(* IEC 61131-3 sources: TA/Tests/RetainTest/FB (part 2) *)

    AUTO1_OUT_ULINT[0] := AUTO1_OUT_ULINT[0] + 1;
    AUTO1_OUT_ULINT[1] := AUTO1_OUT_ULINT[1] + 1;
    AUTO1_OUT_ULINT[2] := AUTO1_OUT_ULINT[2] + 1;
    AUTO1_OUT_ULINT[3] := AUTO1_OUT_ULINT[3] + 1;
    AUTO1_OUT_ULINT[4] := AUTO1_OUT_ULINT[4] + 1;
    AUTO1_OUT_ULINT[5] := AUTO1_OUT_ULINT[5] + 1;
    AUTO1_OUT_ULINT[6] := AUTO1_OUT_ULINT[6] + 1;
    AUTO1_OUT_ULINT[7] := AUTO1_OUT_ULINT[7] + 1;
    AUTO1_OUT_ULINT[8] := AUTO1_OUT_ULINT[8] + 1;
    AUTO1_OUT_ULINT[9] := AUTO1_OUT_ULINT[9] + 1;

    AUTO1_OUT_USINT[0] := AUTO1_OUT_USINT[0] + 1;
    AUTO1_OUT_USINT[1] := AUTO1_OUT_USINT[1] + 1;
    AUTO1_OUT_USINT[2] := AUTO1_OUT_USINT[2] + 1;
    AUTO1_OUT_USINT[3] := AUTO1_OUT_USINT[3] + 1;
    AUTO1_OUT_USINT[4] := AUTO1_OUT_USINT[4] + 1;
    AUTO1_OUT_USINT[5] := AUTO1_OUT_USINT[5] + 1;
    AUTO1_OUT_USINT[6] := AUTO1_OUT_USINT[6] + 1;
    AUTO1_OUT_USINT[7] := AUTO1_OUT_USINT[7] + 1;
    AUTO1_OUT_USINT[8] := AUTO1_OUT_USINT[8] + 1;
    AUTO1_OUT_USINT[9] := AUTO1_OUT_USINT[9] + 1;

    AUTO1_OUT_WORD[0] := AUTO1_OUT_WORD[0] + 1;
    AUTO1_OUT_WORD[1] := AUTO1_OUT_WORD[1] + 1;
    AUTO1_OUT_WORD[2] := AUTO1_OUT_WORD[2] + 1;
    AUTO1_OUT_WORD[3] := AUTO1_OUT_WORD[3] + 1;
    AUTO1_OUT_WORD[4] := AUTO1_OUT_WORD[4] + 1;
    AUTO1_OUT_WORD[5] := AUTO1_OUT_WORD[5] + 1;
    AUTO1_OUT_WORD[6] := AUTO1_OUT_WORD[6] + 1;
    AUTO1_OUT_WORD[7] := AUTO1_OUT_WORD[7] + 1;
    AUTO1_OUT_WORD[8] := AUTO1_OUT_WORD[8] + 1;
    AUTO1_OUT_WORD[9] := AUTO1_OUT_WORD[9] + 1;

    AUTO2_OUT_BOOL[0] := AUTO1_OUT_BOOL[0];
    AUTO2_OUT_BOOL[1] := AUTO1_OUT_BOOL[1];
    AUTO2_OUT_BOOL[2] := AUTO1_OUT_BOOL[2];
    AUTO2_OUT_BOOL[3] := AUTO1_OUT_BOOL[3];
    AUTO2_OUT_BOOL[4] := AUTO1_OUT_BOOL[4];
    AUTO2_OUT_BOOL[5] := AUTO1_OUT_BOOL[5];
    AUTO2_OUT_BOOL[6] := AUTO1_OUT_BOOL[6];
    AUTO2_OUT_BOOL[7] := AUTO1_OUT_BOOL[7];
    AUTO2_OUT_BOOL[8] := AUTO1_OUT_BOOL[8];
    AUTO2_OUT_BOOL[9] := AUTO1_OUT_BOOL[9];

    AUTO2_OUT_BYTE[0] := AUTO1_OUT_BYTE[0];
    AUTO2_OUT_BYTE[1] := AUTO1_OUT_BYTE[1];
    AUTO2_OUT_BYTE[2] := AUTO1_OUT_BYTE[2];
    AUTO2_OUT_BYTE[3] := AUTO1_OUT_BYTE[3];
    AUTO2_OUT_BYTE[4] := AUTO1_OUT_BYTE[4];
    AUTO2_OUT_BYTE[5] := AUTO1_OUT_BYTE[5];
    AUTO2_OUT_BYTE[6] := AUTO1_OUT_BYTE[6];
    AUTO2_OUT_BYTE[7] := AUTO1_OUT_BYTE[7];
    AUTO2_OUT_BYTE[8] := AUTO1_OUT_BYTE[8];
    AUTO2_OUT_BYTE[9] := AUTO1_OUT_BYTE[9];

    AUTO2_OUT_DATE[0] := AUTO1_OUT_DATE[0];
    AUTO2_OUT_DATE[1] := AUTO1_OUT_DATE[1];
    AUTO2_OUT_DATE[2] := AUTO1_OUT_DATE[2];
    AUTO2_OUT_DATE[3] := AUTO1_OUT_DATE[3];
    AUTO2_OUT_DATE[4] := AUTO1_OUT_DATE[4];
    AUTO2_OUT_DATE[5] := AUTO1_OUT_DATE[5];
    AUTO2_OUT_DATE[6] := AUTO1_OUT_DATE[6];
    AUTO2_OUT_DATE[7] := AUTO1_OUT_DATE[7];
    AUTO2_OUT_DATE[8] := AUTO1_OUT_DATE[8];
    AUTO2_OUT_DATE[9] := AUTO1_OUT_DATE[9];

    AUTO2_OUT_DINT[0] := AUTO1_OUT_DINT[0];
    AUTO2_OUT_DINT[1] := AUTO1_OUT_DINT[1];
    AUTO2_OUT_DINT[2] := AUTO1_OUT_DINT[2];
    AUTO2_OUT_DINT[3] := AUTO1_OUT_DINT[3];
    AUTO2_OUT_DINT[4] := AUTO1_OUT_DINT[4];
    AUTO2_OUT_DINT[5] := AUTO1_OUT_DINT[5];
    AUTO2_OUT_DINT[6] := AUTO1_OUT_DINT[6];
    AUTO2_OUT_DINT[7] := AUTO1_OUT_DINT[7];
    AUTO2_OUT_DINT[8] := AUTO1_OUT_DINT[8];
    AUTO2_OUT_DINT[9] := AUTO1_OUT_DINT[9];

    AUTO2_OUT_DWORD[0] := AUTO1_OUT_DWORD[0];
    AUTO2_OUT_DWORD[1] := AUTO1_OUT_DWORD[1];
    AUTO2_OUT_DWORD[2] := AUTO1_OUT_DWORD[2];
    AUTO2_OUT_DWORD[3] := AUTO1_OUT_DWORD[3];
    AUTO2_OUT_DWORD[4] := AUTO1_OUT_DWORD[4];
    AUTO2_OUT_DWORD[5] := AUTO1_OUT_DWORD[5];
    AUTO2_OUT_DWORD[6] := AUTO1_OUT_DWORD[6];
    AUTO2_OUT_DWORD[7] := AUTO1_OUT_DWORD[7];
    AUTO2_OUT_DWORD[8] := AUTO1_OUT_DWORD[8];
    AUTO2_OUT_DWORD[9] := AUTO1_OUT_DWORD[9];

    AUTO2_OUT_INT[0] := AUTO1_OUT_INT[0];
    AUTO2_OUT_INT[1] := AUTO1_OUT_INT[1];
    AUTO2_OUT_INT[2] := AUTO1_OUT_INT[2];
    AUTO2_OUT_INT[3] := AUTO1_OUT_INT[3];
    AUTO2_OUT_INT[4] := AUTO1_OUT_INT[4];
    AUTO2_OUT_INT[5] := AUTO1_OUT_INT[5];
    AUTO2_OUT_INT[6] := AUTO1_OUT_INT[6];
    AUTO2_OUT_INT[7] := AUTO1_OUT_INT[7];
    AUTO2_OUT_INT[8] := AUTO1_OUT_INT[8];
    AUTO2_OUT_INT[9] := AUTO1_OUT_INT[9];

    AUTO2_OUT_LINT[0] := AUTO1_OUT_LINT[0];
    AUTO2_OUT_LINT[1] := AUTO1_OUT_LINT[1];
    AUTO2_OUT_LINT[2] := AUTO1_OUT_LINT[2];
    AUTO2_OUT_LINT[3] := AUTO1_OUT_LINT[3];
    AUTO2_OUT_LINT[4] := AUTO1_OUT_LINT[4];
    AUTO2_OUT_LINT[5] := AUTO1_OUT_LINT[5];
    AUTO2_OUT_LINT[6] := AUTO1_OUT_LINT[6];
    AUTO2_OUT_LINT[7] := AUTO1_OUT_LINT[7];
    AUTO2_OUT_LINT[8] := AUTO1_OUT_LINT[8];
    AUTO2_OUT_LINT[9] := AUTO1_OUT_LINT[9];

    AUTO2_OUT_LREAL[0] := AUTO1_OUT_LREAL[0];
    AUTO2_OUT_LREAL[1] := AUTO1_OUT_LREAL[1];
    AUTO2_OUT_LREAL[2] := AUTO1_OUT_LREAL[2];
    AUTO2_OUT_LREAL[3] := AUTO1_OUT_LREAL[3];
    AUTO2_OUT_LREAL[4] := AUTO1_OUT_LREAL[4];
    AUTO2_OUT_LREAL[5] := AUTO1_OUT_LREAL[5];
    AUTO2_OUT_LREAL[6] := AUTO1_OUT_LREAL[6];
    AUTO2_OUT_LREAL[7] := AUTO1_OUT_LREAL[7];
    AUTO2_OUT_LREAL[8] := AUTO1_OUT_LREAL[8];
    AUTO2_OUT_LREAL[9] := AUTO1_OUT_LREAL[9];

    AUTO2_OUT_LWORD[0] := AUTO1_OUT_LWORD[0];
    AUTO2_OUT_LWORD[1] := AUTO1_OUT_LWORD[1];
    AUTO2_OUT_LWORD[2] := AUTO1_OUT_LWORD[2];
    AUTO2_OUT_LWORD[3] := AUTO1_OUT_LWORD[3];
    AUTO2_OUT_LWORD[4] := AUTO1_OUT_LWORD[4];
    AUTO2_OUT_LWORD[5] := AUTO1_OUT_LWORD[5];
    AUTO2_OUT_LWORD[6] := AUTO1_OUT_LWORD[6];
    AUTO2_OUT_LWORD[7] := AUTO1_OUT_LWORD[7];
    AUTO2_OUT_LWORD[8] := AUTO1_OUT_LWORD[8];
    AUTO2_OUT_LWORD[9] := AUTO1_OUT_LWORD[9];

    AUTO2_OUT_REAL[0] := AUTO1_OUT_REAL[0];
    AUTO2_OUT_REAL[1] := AUTO1_OUT_REAL[1];
    AUTO2_OUT_REAL[2] := AUTO1_OUT_REAL[2];
    AUTO2_OUT_REAL[3] := AUTO1_OUT_REAL[3];
    AUTO2_OUT_REAL[4] := AUTO1_OUT_REAL[4];
    AUTO2_OUT_REAL[5] := AUTO1_OUT_REAL[5];
    AUTO2_OUT_REAL[6] := AUTO1_OUT_REAL[6];
    AUTO2_OUT_REAL[7] := AUTO1_OUT_REAL[7];
    AUTO2_OUT_REAL[8] := AUTO1_OUT_REAL[8];
    AUTO2_OUT_REAL[9] := AUTO1_OUT_REAL[9];

    AUTO2_OUT_SINT[0] := AUTO1_OUT_SINT[0];
    AUTO2_OUT_SINT[1] := AUTO1_OUT_SINT[1];
    AUTO2_OUT_SINT[2] := AUTO1_OUT_SINT[2];
    AUTO2_OUT_SINT[3] := AUTO1_OUT_SINT[3];
    AUTO2_OUT_SINT[4] := AUTO1_OUT_SINT[4];
    AUTO2_OUT_SINT[5] := AUTO1_OUT_SINT[5];
    AUTO2_OUT_SINT[6] := AUTO1_OUT_SINT[6];
    AUTO2_OUT_SINT[7] := AUTO1_OUT_SINT[7];
    AUTO2_OUT_SINT[8] := AUTO1_OUT_SINT[8];
    AUTO2_OUT_SINT[9] := AUTO1_OUT_SINT[9];

    AUTO2_OUT_STRING[0] := AUTO1_OUT_STRING[0];
    AUTO2_OUT_STRING[1] := AUTO1_OUT_STRING[1];
    AUTO2_OUT_STRING[2] := AUTO1_OUT_STRING[2];
    AUTO2_OUT_STRING[3] := AUTO1_OUT_STRING[3];
    AUTO2_OUT_STRING[4] := AUTO1_OUT_STRING[4];
    AUTO2_OUT_STRING[5] := AUTO1_OUT_STRING[5];
    AUTO2_OUT_STRING[6] := AUTO1_OUT_STRING[6];
    AUTO2_OUT_STRING[7] := AUTO1_OUT_STRING[7];
    AUTO2_OUT_STRING[8] := AUTO1_OUT_STRING[8];
    AUTO2_OUT_STRING[9] := AUTO1_OUT_STRING[9];

    AUTO2_OUT_TIME[0] := AUTO1_OUT_TIME[0];
    AUTO2_OUT_TIME[1] := AUTO1_OUT_TIME[1];
    AUTO2_OUT_TIME[2] := AUTO1_OUT_TIME[2];
    AUTO2_OUT_TIME[3] := AUTO1_OUT_TIME[3];
    AUTO2_OUT_TIME[4] := AUTO1_OUT_TIME[4];
    AUTO2_OUT_TIME[5] := AUTO1_OUT_TIME[5];
    AUTO2_OUT_TIME[6] := AUTO1_OUT_TIME[6];
    AUTO2_OUT_TIME[7] := AUTO1_OUT_TIME[7];
    AUTO2_OUT_TIME[8] := AUTO1_OUT_TIME[8];
    AUTO2_OUT_TIME[9] := AUTO1_OUT_TIME[9];

    AUTO2_OUT_UDINT[0] := AUTO1_OUT_UDINT[0];
    AUTO2_OUT_UDINT[1] := AUTO1_OUT_UDINT[1];
    AUTO2_OUT_UDINT[2] := AUTO1_OUT_UDINT[2];
    AUTO2_OUT_UDINT[3] := AUTO1_OUT_UDINT[3];
    AUTO2_OUT_UDINT[4] := AUTO1_OUT_UDINT[4];
    AUTO2_OUT_UDINT[5] := AUTO1_OUT_UDINT[5];
    AUTO2_OUT_UDINT[6] := AUTO1_OUT_UDINT[6];
    AUTO2_OUT_UDINT[7] := AUTO1_OUT_UDINT[7];
    AUTO2_OUT_UDINT[8] := AUTO1_OUT_UDINT[8];
    AUTO2_OUT_UDINT[9] := AUTO1_OUT_UDINT[9];

    AUTO2_OUT_UINT[0] := AUTO1_OUT_UINT[0];
    AUTO2_OUT_UINT[1] := AUTO1_OUT_UINT[1];
    AUTO2_OUT_UINT[2] := AUTO1_OUT_UINT[2];
    AUTO2_OUT_UINT[3] := AUTO1_OUT_UINT[3];
    AUTO2_OUT_UINT[4] := AUTO1_OUT_UINT[4];
    AUTO2_OUT_UINT[5] := AUTO1_OUT_UINT[5];
    AUTO2_OUT_UINT[6] := AUTO1_OUT_UINT[6];
    AUTO2_OUT_UINT[7] := AUTO1_OUT_UINT[7];
    AUTO2_OUT_UINT[8] := AUTO1_OUT_UINT[8];
    AUTO2_OUT_UINT[9] := AUTO1_OUT_UINT[9];

    AUTO2_OUT_ULINT[0] := AUTO1_OUT_ULINT[0];
    AUTO2_OUT_ULINT[1] := AUTO1_OUT_ULINT[1];
    AUTO2_OUT_ULINT[2] := AUTO1_OUT_ULINT[2];
    AUTO2_OUT_ULINT[3] := AUTO1_OUT_ULINT[3];
    AUTO2_OUT_ULINT[4] := AUTO1_OUT_ULINT[4];
    AUTO2_OUT_ULINT[5] := AUTO1_OUT_ULINT[5];
    AUTO2_OUT_ULINT[6] := AUTO1_OUT_ULINT[6];
    AUTO2_OUT_ULINT[7] := AUTO1_OUT_ULINT[7];
    AUTO2_OUT_ULINT[8] := AUTO1_OUT_ULINT[8];
    AUTO2_OUT_ULINT[9] := AUTO1_OUT_ULINT[9];

    AUTO2_OUT_USINT[0] := AUTO1_OUT_USINT[0];
    AUTO2_OUT_USINT[1] := AUTO1_OUT_USINT[1];
    AUTO2_OUT_USINT[2] := AUTO1_OUT_USINT[2];
    AUTO2_OUT_USINT[3] := AUTO1_OUT_USINT[3];
    AUTO2_OUT_USINT[4] := AUTO1_OUT_USINT[4];
    AUTO2_OUT_USINT[5] := AUTO1_OUT_USINT[5];
    AUTO2_OUT_USINT[6] := AUTO1_OUT_USINT[6];
    AUTO2_OUT_USINT[7] := AUTO1_OUT_USINT[7];
    AUTO2_OUT_USINT[8] := AUTO1_OUT_USINT[8];
    AUTO2_OUT_USINT[9] := AUTO1_OUT_USINT[9];

    AUTO2_OUT_WORD[0] := AUTO1_OUT_WORD[0];
    AUTO2_OUT_WORD[1] := AUTO1_OUT_WORD[1];
    AUTO2_OUT_WORD[2] := AUTO1_OUT_WORD[2];
    AUTO2_OUT_WORD[3] := AUTO1_OUT_WORD[3];
    AUTO2_OUT_WORD[4] := AUTO1_OUT_WORD[4];
    AUTO2_OUT_WORD[5] := AUTO1_OUT_WORD[5];
    AUTO2_OUT_WORD[6] := AUTO1_OUT_WORD[6];
    AUTO2_OUT_WORD[7] := AUTO1_OUT_WORD[7];
    AUTO2_OUT_WORD[8] := AUTO1_OUT_WORD[8];
    AUTO2_OUT_WORD[9] := AUTO1_OUT_WORD[9];

END_IF;

END_FUNCTION_BLOCK

(* ---- RetainFbFbSimple.st ---- *)
FUNCTION_BLOCK RetainFbFbSimple

FB_RETAIN(.IN1_BOOL, .IN1_BYTE, .IN1_DATE, .IN1_DINT, .IN1_DWORD, .IN1_INT, .IN1_LINT, .IN1_LREAL, .IN1_LWORD, .IN1_REAL, .IN1_SINT, .IN1_STRING, .IN1_TIME, .IN1_UDINT, .IN1_UINT, .IN1_ULINT, .IN1_USINT, .IN1_WORD, .IN2_BOOL, .IN2_BYTE, .IN2_DATE, .IN2_DINT, .IN2_DWORD, .IN2_INT, .IN2_LINT, .IN2_LREAL, .IN2_LWORD, .IN2_REAL, .IN2_SINT, .IN2_STRING, .IN2_TIME, .IN2_UDINT, .IN2_UINT, .IN2_ULINT, .IN2_USINT, .IN2_WORD, .TRIGGER_IMP, .StartGenerate, .PULSE_TIME);
FB_NONRETAIN(.IN1_BOOL, .IN1_BYTE, .IN1_DATE, .IN1_DINT, .IN1_DWORD, .IN1_INT, .IN1_LINT, .IN1_LREAL, .IN1_LWORD, .IN1_REAL, .IN1_SINT, .IN1_STRING, .IN1_TIME, .IN1_UDINT, .IN1_UINT, .IN1_ULINT, .IN1_USINT, .IN1_WORD, .IN2_BOOL, .IN2_BYTE, .IN2_DATE, .IN2_DINT, .IN2_DWORD, .IN2_INT, .IN2_LINT, .IN2_LREAL, .IN2_LWORD, .IN2_REAL, .IN2_SINT, .IN2_STRING, .IN2_TIME, .IN2_UDINT, .IN2_UINT, .IN2_ULINT, .IN2_USINT, .IN2_WORD, .TRIGGER_IMP, .StartGenerate, .PULSE_TIME);
FB_AUTO(.IN1_BOOL, .IN1_BYTE, .IN1_DATE, .IN1_DINT, .IN1_DWORD, .IN1_INT, .IN1_LINT, .IN1_LREAL, .IN1_LWORD, .IN1_REAL, .IN1_SINT, .IN1_STRING, .IN1_TIME, .IN1_UDINT, .IN1_UINT, .IN1_ULINT, .IN1_USINT, .IN1_WORD, .IN2_BOOL, .IN2_BYTE, .IN2_DATE, .IN2_DINT, .IN2_DWORD, .IN2_INT, .IN2_LINT, .IN2_LREAL, .IN2_LWORD, .IN2_REAL, .IN2_SINT, .IN2_STRING, .IN2_TIME, .IN2_UDINT, .IN2_UINT, .IN2_ULINT, .IN2_USINT, .IN2_WORD, .TRIGGER_IMP, .StartGenerate, .PULSE_TIME);

FB_RETAIN.TRIGGER_IMP := TRIGGER_IMP;
FB_RETAIN.StartGenerate := StartGenerate;
FB_RETAIN.PULSE_TIME := PULSE_TIME;

FB_NONRETAIN.TRIGGER_IMP := TRIGGER_IMP;
FB_NONRETAIN.StartGenerate := StartGenerate;
FB_NONRETAIN.PULSE_TIME := PULSE_TIME;

FB_AUTO.TRIGGER_IMP := TRIGGER_IMP;
FB_AUTO.StartGenerate := StartGenerate;
FB_AUTO.PULSE_TIME := PULSE_TIME;

IF TRIGGER_IMP AND StartGenerate THEN
    FB_RETAIN.IN1_BOOL := NOT FB_RETAIN.IN1_BOOL;
    FB_RETAIN.IN1_BYTE := FB_RETAIN.IN1_BYTE + 1;
    FB_RETAIN.IN1_DATE := ANY_TO_DATE(1445385600 + FB_RETAIN.IN1_DINT * 86400);
    FB_RETAIN.IN1_DINT := FB_RETAIN.IN1_DINT + 1;
    FB_RETAIN.IN1_DWORD := FB_RETAIN.IN1_DWORD + 1;
    FB_RETAIN.IN1_INT := FB_RETAIN.IN1_INT + 1;
    FB_RETAIN.IN1_LINT := FB_RETAIN.IN1_LINT + 1;
    FB_RETAIN.IN1_LREAL := FB_RETAIN.IN1_LREAL + 1.1;
    FB_RETAIN.IN1_LWORD := FB_RETAIN.IN1_LWORD + 1;
    FB_RETAIN.IN1_REAL := FB_RETAIN.IN1_REAL + 1.1;
    FB_RETAIN.IN1_SINT := FB_RETAIN.IN1_SINT + 1;
    FB_RETAIN.IN1_STRING := ANY_TO_STRING(FB_RETAIN.IN1_DINT) + ' ' + ANY_TO_STRING(FB_RETAIN.IN1_TIME);
    FB_RETAIN.IN1_TIME := FB_RETAIN.IN1_TIME + PULSE_TIME;
    FB_RETAIN.IN1_UDINT := FB_RETAIN.IN1_UDINT + 1;
    FB_RETAIN.IN1_UINT := FB_RETAIN.IN1_UINT + 1;
    FB_RETAIN.IN1_ULINT := FB_RETAIN.IN1_ULINT + 1;
    FB_RETAIN.IN1_USINT := FB_RETAIN.IN1_USINT + 1;
    FB_RETAIN.IN1_WORD := FB_RETAIN.IN1_WORD + 1;

    FB_RETAIN.IN2_BOOL := FB_RETAIN.IN1_BOOL;
    FB_RETAIN.IN2_BYTE := FB_RETAIN.IN1_BYTE;
    FB_RETAIN.IN2_DATE := FB_RETAIN.IN1_DATE;
    FB_RETAIN.IN2_DINT := FB_RETAIN.IN1_DINT;
    FB_RETAIN.IN2_DWORD := FB_RETAIN.IN1_DWORD;
    FB_RETAIN.IN2_INT := FB_RETAIN.IN1_INT;
    FB_RETAIN.IN2_LINT := FB_RETAIN.IN1_LINT;
    FB_RETAIN.IN2_LREAL := FB_RETAIN.IN1_LREAL;
    FB_RETAIN.IN2_LWORD := FB_RETAIN.IN1_LWORD;
    FB_RETAIN.IN2_REAL := FB_RETAIN.IN1_REAL;
    FB_RETAIN.IN2_SINT := FB_RETAIN.IN1_SINT;
    FB_RETAIN.IN2_STRING := FB_RETAIN.IN1_STRING;
    FB_RETAIN.IN2_TIME := FB_RETAIN.IN1_TIME;
    FB_RETAIN.IN2_UDINT := FB_RETAIN.IN1_UDINT;
    FB_RETAIN.IN2_UINT := FB_RETAIN.IN1_UINT;
    FB_RETAIN.IN2_ULINT := FB_RETAIN.IN1_ULINT;
    FB_RETAIN.IN2_USINT := FB_RETAIN.IN1_USINT;
    FB_RETAIN.IN2_WORD := FB_RETAIN.IN1_WORD;

    FB_NONRETAIN.IN1_BOOL := NOT FB_NONRETAIN.IN1_BOOL;
    FB_NONRETAIN.IN1_BYTE := FB_NONRETAIN.IN1_BYTE + 1;
    FB_NONRETAIN.IN1_DATE := ANY_TO_DATE(1445385600 + FB_NONRETAIN.IN1_DINT * 86400);
    FB_NONRETAIN.IN1_DINT := FB_NONRETAIN.IN1_DINT + 1;
    FB_NONRETAIN.IN1_DWORD := FB_NONRETAIN.IN1_DWORD + 1;
    FB_NONRETAIN.IN1_INT := FB_NONRETAIN.IN1_INT + 1;
    FB_NONRETAIN.IN1_LINT := FB_NONRETAIN.IN1_LINT + 1;
    FB_NONRETAIN.IN1_LREAL := FB_NONRETAIN.IN1_LREAL + 1.1;
    FB_NONRETAIN.IN1_LWORD := FB_NONRETAIN.IN1_LWORD + 1;
    FB_NONRETAIN.IN1_REAL := FB_NONRETAIN.IN1_REAL + 1.1;
    FB_NONRETAIN.IN1_SINT := FB_NONRETAIN.IN1_SINT + 1;
    FB_NONRETAIN.IN1_STRING := ANY_TO_STRING(FB_NONRETAIN.IN1_DINT) + ' ' + ANY_TO_STRING(FB_NONRETAIN.IN1_TIME);
    FB_NONRETAIN.IN1_TIME := FB_NONRETAIN.IN1_TIME + PULSE_TIME;
    FB_NONRETAIN.IN1_UDINT := FB_NONRETAIN.IN1_UDINT + 1;
    FB_NONRETAIN.IN1_UINT := FB_NONRETAIN.IN1_UINT + 1;
    FB_NONRETAIN.IN1_ULINT := FB_NONRETAIN.IN1_ULINT + 1;
    FB_NONRETAIN.IN1_USINT := FB_NONRETAIN.IN1_USINT + 1;
    FB_NONRETAIN.IN1_WORD := FB_NONRETAIN.IN1_WORD + 1;

    FB_NONRETAIN.IN2_BOOL := FB_NONRETAIN.IN1_BOOL;
    FB_NONRETAIN.IN2_BYTE := FB_NONRETAIN.IN1_BYTE;
    FB_NONRETAIN.IN2_DATE := FB_NONRETAIN.IN1_DATE;
    FB_NONRETAIN.IN2_DINT := FB_NONRETAIN.IN1_DINT;
    FB_NONRETAIN.IN2_DWORD := FB_NONRETAIN.IN1_DWORD;
    FB_NONRETAIN.IN2_INT := FB_NONRETAIN.IN1_INT;
    FB_NONRETAIN.IN2_LINT := FB_NONRETAIN.IN1_LINT;
    FB_NONRETAIN.IN2_LREAL := FB_NONRETAIN.IN1_LREAL;
    FB_NONRETAIN.IN2_LWORD := FB_NONRETAIN.IN1_LWORD;
    FB_NONRETAIN.IN2_REAL := FB_NONRETAIN.IN1_REAL;
    FB_NONRETAIN.IN2_SINT := FB_NONRETAIN.IN1_SINT;
    FB_NONRETAIN.IN2_STRING := FB_NONRETAIN.IN1_STRING;
    FB_NONRETAIN.IN2_TIME := FB_NONRETAIN.IN1_TIME;
    FB_NONRETAIN.IN2_UDINT := FB_NONRETAIN.IN1_UDINT;
    FB_NONRETAIN.IN2_UINT := FB_NONRETAIN.IN1_UINT;
    FB_NONRETAIN.IN2_ULINT := FB_NONRETAIN.IN1_ULINT;
    FB_NONRETAIN.IN2_USINT := FB_NONRETAIN.IN1_USINT;
    FB_NONRETAIN.IN2_WORD := FB_NONRETAIN.IN1_WORD;

    FB_AUTO.IN1_BOOL := NOT FB_AUTO.IN1_BOOL;
    FB_AUTO.IN1_BYTE := FB_AUTO.IN1_BYTE + 1;
    FB_AUTO.IN1_DATE := ANY_TO_DATE(1445385600 + FB_AUTO.IN1_DINT * 86400);
    FB_AUTO.IN1_DINT := FB_AUTO.IN1_DINT + 1;
    FB_AUTO.IN1_DWORD := FB_AUTO.IN1_DWORD + 1;
    FB_AUTO.IN1_INT := FB_AUTO.IN1_INT + 1;
    FB_AUTO.IN1_LINT := FB_AUTO.IN1_LINT + 1;
    FB_AUTO.IN1_LREAL := FB_AUTO.IN1_LREAL + 1.1;
    FB_AUTO.IN1_LWORD := FB_AUTO.IN1_LWORD + 1;
    FB_AUTO.IN1_REAL := FB_AUTO.IN1_REAL + 1.1;
    FB_AUTO.IN1_SINT := FB_AUTO.IN1_SINT + 1;
    FB_AUTO.IN1_STRING := ANY_TO_STRING(FB_AUTO.IN1_DINT) + ' ' + ANY_TO_STRING(FB_AUTO.IN1_TIME);
    FB_AUTO.IN1_TIME := FB_AUTO.IN1_TIME + PULSE_TIME;
    FB_AUTO.IN1_UDINT := FB_AUTO.IN1_UDINT + 1;
    FB_AUTO.IN1_UINT := FB_AUTO.IN1_UINT + 1;
    FB_AUTO.IN1_ULINT := FB_AUTO.IN1_ULINT + 1;
    FB_AUTO.IN1_USINT := FB_AUTO.IN1_USINT + 1;
    FB_AUTO.IN1_WORD := FB_AUTO.IN1_WORD + 1;

    FB_AUTO.IN2_BOOL := FB_AUTO.IN1_BOOL;
    FB_AUTO.IN2_BYTE := FB_AUTO.IN1_BYTE;
    FB_AUTO.IN2_DATE := FB_AUTO.IN1_DATE;
    FB_AUTO.IN2_DINT := FB_AUTO.IN1_DINT;
    FB_AUTO.IN2_DWORD := FB_AUTO.IN1_DWORD;
    FB_AUTO.IN2_INT := FB_AUTO.IN1_INT;
    FB_AUTO.IN2_LINT := FB_AUTO.IN1_LINT;
    FB_AUTO.IN2_LREAL := FB_AUTO.IN1_LREAL;
    FB_AUTO.IN2_LWORD := FB_AUTO.IN1_LWORD;
    FB_AUTO.IN2_REAL := FB_AUTO.IN1_REAL;
    FB_AUTO.IN2_SINT := FB_AUTO.IN1_SINT;
    FB_AUTO.IN2_STRING := FB_AUTO.IN1_STRING;
    FB_AUTO.IN2_TIME := FB_AUTO.IN1_TIME;
    FB_AUTO.IN2_UDINT := FB_AUTO.IN1_UDINT;
    FB_AUTO.IN2_UINT := FB_AUTO.IN1_UINT;
    FB_AUTO.IN2_ULINT := FB_AUTO.IN1_ULINT;
    FB_AUTO.IN2_USINT := FB_AUTO.IN1_USINT;
    FB_AUTO.IN2_WORD := FB_AUTO.IN1_WORD;
END_IF;

END_FUNCTION_BLOCK

(* ---- RetainFbSimple.st ---- *)
FUNCTION_BLOCK RetainFbSimple

IF TRIGGER_IMP AND StartGenerate THEN
    RETAIN_LOCAL_BOOL := NOT RETAIN_LOCAL_BOOL;
    RETAIN_LOCAL_BYTE := RETAIN_LOCAL_BYTE + 1;
    RETAIN_LOCAL_DATE := ANY_TO_DATE(1445385600 + RETAIN_LOCAL_DINT * 86400);
    RETAIN_LOCAL_DINT := RETAIN_LOCAL_DINT + 1;
    RETAIN_LOCAL_DWORD := RETAIN_LOCAL_DWORD + 1;
    RETAIN_LOCAL_INT := RETAIN_LOCAL_INT + 1;
    RETAIN_LOCAL_LINT := RETAIN_LOCAL_LINT + 1;
    RETAIN_LOCAL_LREAL := RETAIN_LOCAL_LREAL + 1.1;
    RETAIN_LOCAL_LWORD := RETAIN_LOCAL_LWORD + 1;
    RETAIN_LOCAL_REAL := RETAIN_LOCAL_REAL + 1.1;
    RETAIN_LOCAL_SINT := RETAIN_LOCAL_SINT + 1;
    RETAIN_LOCAL_STRING := ANY_TO_STRING(RETAIN_LOCAL_DINT) + ' ' + ANY_TO_STRING(RETAIN_LOCAL_TIME);
    RETAIN_LOCAL_TIME := RETAIN_LOCAL_TIME + PULSE_TIME;
    RETAIN_LOCAL_UDINT := RETAIN_LOCAL_UDINT + 1;
    RETAIN_LOCAL_UINT := RETAIN_LOCAL_UINT + 1;
    RETAIN_LOCAL_ULINT := RETAIN_LOCAL_ULINT + 1;
    RETAIN_LOCAL_USINT := RETAIN_LOCAL_USINT + 1;
    RETAIN_LOCAL_WORD := RETAIN_LOCAL_WORD + 1;

    NONRETAIN_LOCAL_BOOL := NOT NONRETAIN_LOCAL_BOOL;
    NONRETAIN_LOCAL_BYTE := NONRETAIN_LOCAL_BYTE + 1;
    NONRETAIN_LOCAL_DATE := ANY_TO_DATE(1445385600 + NONRETAIN_LOCAL_DINT * 86400);
    NONRETAIN_LOCAL_DINT := NONRETAIN_LOCAL_DINT + 1;
    NONRETAIN_LOCAL_DWORD := NONRETAIN_LOCAL_DWORD + 1;
    NONRETAIN_LOCAL_INT := NONRETAIN_LOCAL_INT + 1;
    NONRETAIN_LOCAL_LINT := NONRETAIN_LOCAL_LINT + 1;
    NONRETAIN_LOCAL_LREAL := NONRETAIN_LOCAL_LREAL + 1.1;
    NONRETAIN_LOCAL_LWORD := NONRETAIN_LOCAL_LWORD + 1;
    NONRETAIN_LOCAL_REAL := NONRETAIN_LOCAL_REAL + 1.1;
    NONRETAIN_LOCAL_SINT := NONRETAIN_LOCAL_SINT + 1;
    NONRETAIN_LOCAL_STRING := ANY_TO_STRING(NONRETAIN_LOCAL_DINT) + ' ' + ANY_TO_STRING(NONRETAIN_LOCAL_TIME);
    NONRETAIN_LOCAL_TIME := NONRETAIN_LOCAL_TIME + PULSE_TIME;
    NONRETAIN_LOCAL_UDINT := NONRETAIN_LOCAL_UDINT + 1;
    NONRETAIN_LOCAL_UINT := NONRETAIN_LOCAL_UINT + 1;
    NONRETAIN_LOCAL_ULINT := NONRETAIN_LOCAL_ULINT + 1;
    NONRETAIN_LOCAL_USINT := NONRETAIN_LOCAL_USINT + 1;
    NONRETAIN_LOCAL_WORD := NONRETAIN_LOCAL_WORD + 1;

    AUTO1_LOCAL_BOOL := NOT AUTO1_LOCAL_BOOL;
    AUTO1_LOCAL_BYTE := AUTO1_LOCAL_BYTE + 1;
    AUTO1_LOCAL_DATE := ANY_TO_DATE(1445385600 + AUTO1_LOCAL_DINT * 86400);
    AUTO1_LOCAL_DINT := AUTO1_LOCAL_DINT + 1;
    AUTO1_LOCAL_DWORD := AUTO1_LOCAL_DWORD + 1;
    AUTO1_LOCAL_INT := AUTO1_LOCAL_INT + 1;
    AUTO1_LOCAL_LINT := AUTO1_LOCAL_LINT + 1;
    AUTO1_LOCAL_LREAL := AUTO1_LOCAL_LREAL + 1.1;
    AUTO1_LOCAL_LWORD := AUTO1_LOCAL_LWORD + 1;
    AUTO1_LOCAL_REAL := AUTO1_LOCAL_REAL + 1.1;
    AUTO1_LOCAL_SINT := AUTO1_LOCAL_SINT + 1;
    AUTO1_LOCAL_STRING := ANY_TO_STRING(AUTO1_LOCAL_DINT) + ' ' + ANY_TO_STRING(AUTO1_LOCAL_TIME);
    AUTO1_LOCAL_TIME := AUTO1_LOCAL_TIME + PULSE_TIME;
    AUTO1_LOCAL_UDINT := AUTO1_LOCAL_UDINT + 1;
    AUTO1_LOCAL_UINT := AUTO1_LOCAL_UINT + 1;
    AUTO1_LOCAL_ULINT := AUTO1_LOCAL_ULINT + 1;
    AUTO1_LOCAL_USINT := AUTO1_LOCAL_USINT + 1;
    AUTO1_LOCAL_WORD := AUTO1_LOCAL_WORD + 1;

    AUTO2_LOCAL_BOOL := AUTO1_LOCAL_BOOL;
    AUTO2_LOCAL_BYTE := AUTO1_LOCAL_BYTE;
    AUTO2_LOCAL_DATE := AUTO1_LOCAL_DATE;
    AUTO2_LOCAL_DINT := AUTO1_LOCAL_DINT;
    AUTO2_LOCAL_DWORD := AUTO1_LOCAL_DWORD;
    AUTO2_LOCAL_INT := AUTO1_LOCAL_INT;
    AUTO2_LOCAL_LINT := AUTO1_LOCAL_LINT;
    AUTO2_LOCAL_LREAL := AUTO1_LOCAL_LREAL;
    AUTO2_LOCAL_LWORD := AUTO1_LOCAL_LWORD;
    AUTO2_LOCAL_REAL := AUTO1_LOCAL_REAL;
    AUTO2_LOCAL_SINT := AUTO1_LOCAL_SINT;
    AUTO2_LOCAL_STRING := AUTO1_LOCAL_STRING;
    AUTO2_LOCAL_TIME := AUTO1_LOCAL_TIME;
    AUTO2_LOCAL_UDINT := AUTO1_LOCAL_UDINT;
    AUTO2_LOCAL_UINT := AUTO1_LOCAL_UINT;
    AUTO2_LOCAL_ULINT := AUTO1_LOCAL_ULINT;
    AUTO2_LOCAL_USINT := AUTO1_LOCAL_USINT;
    AUTO2_LOCAL_WORD := AUTO1_LOCAL_WORD;

    RETAIN_OUT_BOOL := NOT RETAIN_OUT_BOOL;
    RETAIN_OUT_BYTE := RETAIN_OUT_BYTE + 1;
    RETAIN_OUT_DATE := ANY_TO_DATE(1445385600 + RETAIN_OUT_DINT * 86400);
    RETAIN_OUT_DINT := RETAIN_OUT_DINT + 1;
    RETAIN_OUT_DWORD := RETAIN_OUT_DWORD + 1;
    RETAIN_OUT_INT := RETAIN_OUT_INT + 1;
    RETAIN_OUT_LINT := RETAIN_OUT_LINT + 1;
    RETAIN_OUT_LREAL := RETAIN_OUT_LREAL + 1.1;
    RETAIN_OUT_LWORD := RETAIN_OUT_LWORD + 1;
    RETAIN_OUT_REAL := RETAIN_OUT_REAL + 1.1;
    RETAIN_OUT_SINT := RETAIN_OUT_SINT + 1;
    RETAIN_OUT_STRING := ANY_TO_STRING(RETAIN_OUT_DINT) + ' ' + ANY_TO_STRING(RETAIN_OUT_TIME);
    RETAIN_OUT_TIME := RETAIN_OUT_TIME + PULSE_TIME;
    RETAIN_OUT_UDINT := RETAIN_OUT_UDINT + 1;
    RETAIN_OUT_UINT := RETAIN_OUT_UINT + 1;
    RETAIN_OUT_ULINT := RETAIN_OUT_ULINT + 1;
    RETAIN_OUT_USINT := RETAIN_OUT_USINT + 1;
    RETAIN_OUT_WORD := RETAIN_OUT_WORD + 1;

    NONRETAIN_OUT_BOOL := NOT NONRETAIN_OUT_BOOL;
    NONRETAIN_OUT_BYTE := NONRETAIN_OUT_BYTE + 1;
    NONRETAIN_OUT_DATE := ANY_TO_DATE(1445385600 + NONRETAIN_OUT_DINT * 86400);
    NONRETAIN_OUT_DINT := NONRETAIN_OUT_DINT + 1;
    NONRETAIN_OUT_DWORD := NONRETAIN_OUT_DWORD + 1;
    NONRETAIN_OUT_INT := NONRETAIN_OUT_INT + 1;
    NONRETAIN_OUT_LINT := NONRETAIN_OUT_LINT + 1;
    NONRETAIN_OUT_LREAL := NONRETAIN_OUT_LREAL + 1.1;
    NONRETAIN_OUT_LWORD := NONRETAIN_OUT_LWORD + 1;
    NONRETAIN_OUT_REAL := NONRETAIN_OUT_REAL + 1.1;
    NONRETAIN_OUT_SINT := NONRETAIN_OUT_SINT + 1;
    NONRETAIN_OUT_STRING := ANY_TO_STRING(NONRETAIN_OUT_DINT) + ' ' + ANY_TO_STRING(NONRETAIN_OUT_TIME);
    NONRETAIN_OUT_TIME := NONRETAIN_OUT_TIME + PULSE_TIME;
    NONRETAIN_OUT_UDINT := NONRETAIN_OUT_UDINT + 1;
    NONRETAIN_OUT_UINT := NONRETAIN_OUT_UINT + 1;
    NONRETAIN_OUT_ULINT := NONRETAIN_OUT_ULINT + 1;
    NONRETAIN_OUT_USINT := NONRETAIN_OUT_USINT + 1;
    NONRETAIN_OUT_WORD := NONRETAIN_OUT_WORD + 1;

    AUTO1_OUT_BOOL := NOT AUTO1_OUT_BOOL;
    AUTO1_OUT_BYTE := AUTO1_OUT_BYTE + 1;
    AUTO1_OUT_DATE := ANY_TO_DATE(1445385600 + AUTO1_OUT_DINT * 86400);
    AUTO1_OUT_DINT := AUTO1_OUT_DINT + 1;
    AUTO1_OUT_DWORD := AUTO1_OUT_DWORD + 1;
    AUTO1_OUT_INT := AUTO1_OUT_INT + 1;
    AUTO1_OUT_LINT := AUTO1_OUT_LINT + 1;
    AUTO1_OUT_LREAL := AUTO1_OUT_LREAL + 1.1;
    AUTO1_OUT_LWORD := AUTO1_OUT_LWORD + 1;
    AUTO1_OUT_REAL := AUTO1_OUT_REAL + 1.1;
    AUTO1_OUT_SINT := AUTO1_OUT_SINT + 1;
    AUTO1_OUT_STRING := ANY_TO_STRING(AUTO1_OUT_DINT) + ' ' + ANY_TO_STRING(AUTO1_OUT_TIME);
    AUTO1_OUT_TIME := AUTO1_OUT_TIME + PULSE_TIME;
    AUTO1_OUT_UDINT := AUTO1_OUT_UDINT + 1;
    AUTO1_OUT_UINT := AUTO1_OUT_UINT + 1;
    AUTO1_OUT_ULINT := AUTO1_OUT_ULINT + 1;
    AUTO1_OUT_USINT := AUTO1_OUT_USINT + 1;
    AUTO1_OUT_WORD := AUTO1_OUT_WORD + 1;

    AUTO2_OUT_BOOL := AUTO1_OUT_BOOL;
    AUTO2_OUT_BYTE := AUTO1_OUT_BYTE;
    AUTO2_OUT_DATE := AUTO1_OUT_DATE;
    AUTO2_OUT_DINT := AUTO1_OUT_DINT;
    AUTO2_OUT_DWORD := AUTO1_OUT_DWORD;
    AUTO2_OUT_INT := AUTO1_OUT_INT;
    AUTO2_OUT_LINT := AUTO1_OUT_LINT;
    AUTO2_OUT_LREAL := AUTO1_OUT_LREAL;
    AUTO2_OUT_LWORD := AUTO1_OUT_LWORD;
    AUTO2_OUT_REAL := AUTO1_OUT_REAL;
    AUTO2_OUT_SINT := AUTO1_OUT_SINT;
    AUTO2_OUT_STRING := AUTO1_OUT_STRING;
    AUTO2_OUT_TIME := AUTO1_OUT_TIME;
    AUTO2_OUT_UDINT := AUTO1_OUT_UDINT;
    AUTO2_OUT_UINT := AUTO1_OUT_UINT;
    AUTO2_OUT_ULINT := AUTO1_OUT_ULINT;
    AUTO2_OUT_USINT := AUTO1_OUT_USINT;
    AUTO2_OUT_WORD := AUTO1_OUT_WORD;
END_IF;

END_FUNCTION_BLOCK

(* ---- RetainFbSimpleAuto.st ---- *)
FUNCTION_BLOCK RetainFbSimpleAuto

IF TRIGGER_IMP AND StartGenerate THEN
    LOCAL1_BOOL := NOT LOCAL1_BOOL;
    LOCAL1_BYTE := LOCAL1_BYTE + 1;
    LOCAL1_DATE := ANY_TO_DATE(1445385600 + LOCAL1_DINT * 86400);
    LOCAL1_DINT := LOCAL1_DINT + 1;
    LOCAL1_DWORD := LOCAL1_DWORD + 1;
    LOCAL1_INT := LOCAL1_INT + 1;
    LOCAL1_LINT := LOCAL1_LINT + 1;
    LOCAL1_LREAL := LOCAL1_LREAL + 1.1;
    LOCAL1_LWORD := LOCAL1_LWORD + 1;
    LOCAL1_REAL := LOCAL1_REAL + 1.1;
    LOCAL1_SINT := LOCAL1_SINT + 1;
    LOCAL1_STRING := ANY_TO_STRING(LOCAL1_DINT) + ' ' + ANY_TO_STRING(LOCAL1_TIME);
    LOCAL1_TIME := LOCAL1_TIME + PULSE_TIME;
    LOCAL1_UDINT := LOCAL1_UDINT + 1;
    LOCAL1_UINT := LOCAL1_UINT + 1;
    LOCAL1_ULINT := LOCAL1_ULINT + 1;
    LOCAL1_USINT := LOCAL1_USINT + 1;
    LOCAL1_WORD := LOCAL1_WORD + 1;

    LOCAL2_BOOL := LOCAL1_BOOL;
    LOCAL2_BYTE := LOCAL1_BYTE;
    LOCAL2_DATE := LOCAL1_DATE;
    LOCAL2_DINT := LOCAL1_DINT;
    LOCAL2_DWORD := LOCAL1_DWORD;
    LOCAL2_INT := LOCAL1_INT;
    LOCAL2_LINT := LOCAL1_LINT;
    LOCAL2_LREAL := LOCAL1_LREAL;
    LOCAL2_LWORD := LOCAL1_LWORD;
    LOCAL2_REAL := LOCAL1_REAL;
    LOCAL2_SINT := LOCAL1_SINT;
    LOCAL2_STRING := LOCAL1_STRING;
    LOCAL2_TIME := LOCAL1_TIME;
    LOCAL2_UDINT := LOCAL1_UDINT;
    LOCAL2_UINT := LOCAL1_UINT;
    LOCAL2_ULINT := LOCAL1_ULINT;
    LOCAL2_USINT := LOCAL1_USINT;
    LOCAL2_WORD := LOCAL1_WORD;

    OUT1_BOOL := NOT OUT1_BOOL;
    OUT1_BYTE := OUT1_BYTE + 1;
    OUT1_DATE := ANY_TO_DATE(1445385600 + OUT1_DINT * 86400);
    OUT1_DINT := OUT1_DINT + 1;
    OUT1_DWORD := OUT1_DWORD + 1;
    OUT1_INT := OUT1_INT + 1;
    OUT1_LINT := OUT1_LINT + 1;
    OUT1_LREAL := OUT1_LREAL + 1.1;
    OUT1_LWORD := OUT1_LWORD + 1;
    OUT1_REAL := OUT1_REAL + 1.1;
    OUT1_SINT := OUT1_SINT + 1;
    OUT1_STRING := ANY_TO_STRING(OUT1_DINT) + ' ' + ANY_TO_STRING(OUT1_TIME);
    OUT1_TIME := OUT1_TIME + PULSE_TIME;
    OUT1_UDINT := OUT1_UDINT + 1;
    OUT1_UINT := OUT1_UINT + 1;
    OUT1_ULINT := OUT1_ULINT + 1;
    OUT1_USINT := OUT1_USINT + 1;
    OUT1_WORD := OUT1_WORD + 1;

    OUT2_BOOL := OUT1_BOOL;
    OUT2_BYTE := OUT1_BYTE;
    OUT2_DATE := OUT1_DATE;
    OUT2_DINT := OUT1_DINT;
    OUT2_DWORD := OUT1_DWORD;
    OUT2_INT := OUT1_INT;
    OUT2_LINT := OUT1_LINT;
    OUT2_LREAL := OUT1_LREAL;
    OUT2_LWORD := OUT1_LWORD;
    OUT2_REAL := OUT1_REAL;
    OUT2_SINT := OUT1_SINT;
    OUT2_STRING := OUT1_STRING;
    OUT2_TIME := OUT1_TIME;
    OUT2_UDINT := OUT1_UDINT;
    OUT2_UINT := OUT1_UINT;
    OUT2_ULINT := OUT1_ULINT;
    OUT2_USINT := OUT1_USINT;
    OUT2_WORD := OUT1_WORD;
END_IF;

END_FUNCTION_BLOCK

(* ---- RetainFbStructureSimple.st ---- *)
FUNCTION_BLOCK RetainFbStructureSimple

IF TRIGGER_IMP AND StartGenerate THEN
    RETAIN_LOCAL.SIMPLE_BOOL := NOT RETAIN_LOCAL.SIMPLE_BOOL;
    RETAIN_LOCAL.SIMPLE_BYTE := RETAIN_LOCAL.SIMPLE_BYTE + 1;
    RETAIN_LOCAL.SIMPLE_DATE := ANY_TO_DATE(1445385600 + RETAIN_LOCAL.SIMPLE_DINT * 86400);
    RETAIN_LOCAL.SIMPLE_DINT := RETAIN_LOCAL.SIMPLE_DINT + 1;
    RETAIN_LOCAL.SIMPLE_DWORD := RETAIN_LOCAL.SIMPLE_DWORD + 1;
    RETAIN_LOCAL.SIMPLE_INT := RETAIN_LOCAL.SIMPLE_INT + 1;
    RETAIN_LOCAL.SIMPLE_LINT := RETAIN_LOCAL.SIMPLE_LINT + 1;
    RETAIN_LOCAL.SIMPLE_LREAL := RETAIN_LOCAL.SIMPLE_LREAL + 1.1;
    RETAIN_LOCAL.SIMPLE_LWORD := RETAIN_LOCAL.SIMPLE_LWORD + 1;
    RETAIN_LOCAL.SIMPLE_REAL := RETAIN_LOCAL.SIMPLE_REAL + 1.1;
    RETAIN_LOCAL.SIMPLE_SINT := RETAIN_LOCAL.SIMPLE_SINT + 1;
    RETAIN_LOCAL.SIMPLE_STRING := ANY_TO_STRING(RETAIN_LOCAL.SIMPLE_DINT) + ' ' + ANY_TO_STRING(RETAIN_LOCAL.SIMPLE_TIME);
    RETAIN_LOCAL.SIMPLE_TIME := RETAIN_LOCAL.SIMPLE_TIME + PULSE_TIME;
    RETAIN_LOCAL.SIMPLE_UDINT := RETAIN_LOCAL.SIMPLE_UDINT + 1;
    RETAIN_LOCAL.SIMPLE_UINT := RETAIN_LOCAL.SIMPLE_UINT + 1;
    RETAIN_LOCAL.SIMPLE_ULINT := RETAIN_LOCAL.SIMPLE_ULINT + 1;
    RETAIN_LOCAL.SIMPLE_ULINT := RETAIN_LOCAL.SIMPLE_ULINT + 1;
    RETAIN_LOCAL.SIMPLE_WORD := RETAIN_LOCAL.SIMPLE_WORD + 1;

    NONRETAIN_LOCAL.SIMPLE_BOOL := NOT NONRETAIN_LOCAL.SIMPLE_BOOL;
    NONRETAIN_LOCAL.SIMPLE_BYTE := NONRETAIN_LOCAL.SIMPLE_BYTE + 1;
    NONRETAIN_LOCAL.SIMPLE_DATE := ANY_TO_DATE(1445385600 + NONRETAIN_LOCAL.SIMPLE_DINT * 86400);
    NONRETAIN_LOCAL.SIMPLE_DINT := NONRETAIN_LOCAL.SIMPLE_DINT + 1;
    NONRETAIN_LOCAL.SIMPLE_DWORD := NONRETAIN_LOCAL.SIMPLE_DWORD + 1;
    NONRETAIN_LOCAL.SIMPLE_INT := NONRETAIN_LOCAL.SIMPLE_INT + 1;
    NONRETAIN_LOCAL.SIMPLE_LINT := NONRETAIN_LOCAL.SIMPLE_LINT + 1;
    NONRETAIN_LOCAL.SIMPLE_LREAL := NONRETAIN_LOCAL.SIMPLE_LREAL + 1.1;
    NONRETAIN_LOCAL.SIMPLE_LWORD := NONRETAIN_LOCAL.SIMPLE_LWORD + 1;
    NONRETAIN_LOCAL.SIMPLE_REAL := NONRETAIN_LOCAL.SIMPLE_REAL + 1.1;
    NONRETAIN_LOCAL.SIMPLE_SINT := NONRETAIN_LOCAL.SIMPLE_SINT + 1;
    NONRETAIN_LOCAL.SIMPLE_STRING := ANY_TO_STRING(NONRETAIN_LOCAL.SIMPLE_DINT) + ' ' + ANY_TO_STRING(NONRETAIN_LOCAL.SIMPLE_TIME);
    NONRETAIN_LOCAL.SIMPLE_TIME := NONRETAIN_LOCAL.SIMPLE_TIME + PULSE_TIME;
    NONRETAIN_LOCAL.SIMPLE_UDINT := NONRETAIN_LOCAL.SIMPLE_UDINT + 1;
    NONRETAIN_LOCAL.SIMPLE_UINT := NONRETAIN_LOCAL.SIMPLE_UINT + 1;
    NONRETAIN_LOCAL.SIMPLE_ULINT := NONRETAIN_LOCAL.SIMPLE_ULINT + 1;
    NONRETAIN_LOCAL.SIMPLE_ULINT := NONRETAIN_LOCAL.SIMPLE_ULINT + 1;
    NONRETAIN_LOCAL.SIMPLE_WORD := NONRETAIN_LOCAL.SIMPLE_WORD + 1;

    AUTO1_LOCAL.SIMPLE_BOOL := NOT AUTO1_LOCAL.SIMPLE_BOOL;
    AUTO1_LOCAL.SIMPLE_BYTE := AUTO1_LOCAL.SIMPLE_BYTE + 1;
    AUTO1_LOCAL.SIMPLE_DATE := ANY_TO_DATE(1445385600 + AUTO1_LOCAL.SIMPLE_DINT * 86400);
    AUTO1_LOCAL.SIMPLE_DINT := AUTO1_LOCAL.SIMPLE_DINT + 1;
    AUTO1_LOCAL.SIMPLE_DWORD := AUTO1_LOCAL.SIMPLE_DWORD + 1;
    AUTO1_LOCAL.SIMPLE_INT := AUTO1_LOCAL.SIMPLE_INT + 1;
    AUTO1_LOCAL.SIMPLE_LINT := AUTO1_LOCAL.SIMPLE_LINT + 1;
    AUTO1_LOCAL.SIMPLE_LREAL := AUTO1_LOCAL.SIMPLE_LREAL + 1.1;
    AUTO1_LOCAL.SIMPLE_LWORD := AUTO1_LOCAL.SIMPLE_LWORD + 1;
    AUTO1_LOCAL.SIMPLE_REAL := AUTO1_LOCAL.SIMPLE_REAL + 1.1;
    AUTO1_LOCAL.SIMPLE_SINT := AUTO1_LOCAL.SIMPLE_SINT + 1;
    AUTO1_LOCAL.SIMPLE_STRING := ANY_TO_STRING(AUTO1_LOCAL.SIMPLE_DINT) + ' ' + ANY_TO_STRING(AUTO1_LOCAL.SIMPLE_TIME);
    AUTO1_LOCAL.SIMPLE_TIME := AUTO1_LOCAL.SIMPLE_TIME + PULSE_TIME;
    AUTO1_LOCAL.SIMPLE_UDINT := AUTO1_LOCAL.SIMPLE_UDINT + 1;
    AUTO1_LOCAL.SIMPLE_UINT := AUTO1_LOCAL.SIMPLE_UINT + 1;
    AUTO1_LOCAL.SIMPLE_ULINT := AUTO1_LOCAL.SIMPLE_ULINT + 1;
    AUTO1_LOCAL.SIMPLE_ULINT := AUTO1_LOCAL.SIMPLE_ULINT + 1;
    AUTO1_LOCAL.SIMPLE_WORD := AUTO1_LOCAL.SIMPLE_WORD + 1;

    AUTO2_LOCAL.SIMPLE_BOOL := AUTO1_LOCAL.SIMPLE_BOOL;
    AUTO2_LOCAL.SIMPLE_BYTE := AUTO1_LOCAL.SIMPLE_BYTE;
    AUTO2_LOCAL.SIMPLE_DATE := AUTO1_LOCAL.SIMPLE_DATE;
    AUTO2_LOCAL.SIMPLE_DINT := AUTO1_LOCAL.SIMPLE_DINT;
    AUTO2_LOCAL.SIMPLE_DWORD := AUTO1_LOCAL.SIMPLE_DWORD;
    AUTO2_LOCAL.SIMPLE_INT := AUTO1_LOCAL.SIMPLE_INT;
    AUTO2_LOCAL.SIMPLE_LINT := AUTO1_LOCAL.SIMPLE_LINT;
    AUTO2_LOCAL.SIMPLE_LREAL := AUTO1_LOCAL.SIMPLE_LREAL;
    AUTO2_LOCAL.SIMPLE_LWORD := AUTO1_LOCAL.SIMPLE_LWORD;
    AUTO2_LOCAL.SIMPLE_REAL := AUTO1_LOCAL.SIMPLE_REAL;
    AUTO2_LOCAL.SIMPLE_SINT := AUTO1_LOCAL.SIMPLE_SINT;
    AUTO2_LOCAL.SIMPLE_STRING := AUTO1_LOCAL.SIMPLE_STRING;
    AUTO2_LOCAL.SIMPLE_TIME := AUTO1_LOCAL.SIMPLE_TIME;
    AUTO2_LOCAL.SIMPLE_UDINT := AUTO1_LOCAL.SIMPLE_UDINT;
    AUTO2_LOCAL.SIMPLE_UINT := AUTO1_LOCAL.SIMPLE_UINT;
    AUTO2_LOCAL.SIMPLE_ULINT := AUTO1_LOCAL.SIMPLE_ULINT;
    AUTO2_LOCAL.SIMPLE_ULINT := AUTO1_LOCAL.SIMPLE_ULINT;
    AUTO2_LOCAL.SIMPLE_WORD := AUTO1_LOCAL.SIMPLE_WORD;

    RETAIN_OUT.SIMPLE_BOOL := NOT RETAIN_OUT.SIMPLE_BOOL;
    RETAIN_OUT.SIMPLE_BYTE := RETAIN_OUT.SIMPLE_BYTE + 1;
    RETAIN_OUT.SIMPLE_DATE := ANY_TO_DATE(1445385600 + RETAIN_OUT.SIMPLE_DINT * 86400);
    RETAIN_OUT.SIMPLE_DINT := RETAIN_OUT.SIMPLE_DINT + 1;
    RETAIN_OUT.SIMPLE_DWORD := RETAIN_OUT.SIMPLE_DWORD + 1;
    RETAIN_OUT.SIMPLE_INT := RETAIN_OUT.SIMPLE_INT + 1;
    RETAIN_OUT.SIMPLE_LINT := RETAIN_OUT.SIMPLE_LINT + 1;
    RETAIN_OUT.SIMPLE_LREAL := RETAIN_OUT.SIMPLE_LREAL + 1.1;
    RETAIN_OUT.SIMPLE_LWORD := RETAIN_OUT.SIMPLE_LWORD + 1;
    RETAIN_OUT.SIMPLE_REAL := RETAIN_OUT.SIMPLE_REAL + 1.1;
    RETAIN_OUT.SIMPLE_SINT := RETAIN_OUT.SIMPLE_SINT + 1;
    RETAIN_OUT.SIMPLE_STRING := ANY_TO_STRING(RETAIN_OUT.SIMPLE_DINT) + ' ' + ANY_TO_STRING(RETAIN_OUT.SIMPLE_TIME);
    RETAIN_OUT.SIMPLE_TIME := RETAIN_OUT.SIMPLE_TIME + PULSE_TIME;
    RETAIN_OUT.SIMPLE_UDINT := RETAIN_OUT.SIMPLE_UDINT + 1;
    RETAIN_OUT.SIMPLE_UINT := RETAIN_OUT.SIMPLE_UINT + 1;
    RETAIN_OUT.SIMPLE_ULINT := RETAIN_OUT.SIMPLE_ULINT + 1;
    RETAIN_OUT.SIMPLE_ULINT := RETAIN_OUT.SIMPLE_ULINT + 1;
    RETAIN_OUT.SIMPLE_WORD := RETAIN_OUT.SIMPLE_WORD + 1;

    NONRETAIN_OUT.SIMPLE_BOOL := NOT NONRETAIN_OUT.SIMPLE_BOOL;
    NONRETAIN_OUT.SIMPLE_BYTE := NONRETAIN_OUT.SIMPLE_BYTE + 1;
    NONRETAIN_OUT.SIMPLE_DATE := ANY_TO_DATE(1445385600 + NONRETAIN_OUT.SIMPLE_DINT * 86400);
    NONRETAIN_OUT.SIMPLE_DINT := NONRETAIN_OUT.SIMPLE_DINT + 1;
    NONRETAIN_OUT.SIMPLE_DWORD := NONRETAIN_OUT.SIMPLE_DWORD + 1;
    NONRETAIN_OUT.SIMPLE_INT := NONRETAIN_OUT.SIMPLE_INT + 1;
    NONRETAIN_OUT.SIMPLE_LINT := NONRETAIN_OUT.SIMPLE_LINT + 1;
    NONRETAIN_OUT.SIMPLE_LREAL := NONRETAIN_OUT.SIMPLE_LREAL + 1.1;
    NONRETAIN_OUT.SIMPLE_LWORD := NONRETAIN_OUT.SIMPLE_LWORD + 1;
    NONRETAIN_OUT.SIMPLE_REAL := NONRETAIN_OUT.SIMPLE_REAL + 1.1;
    NONRETAIN_OUT.SIMPLE_SINT := NONRETAIN_OUT.SIMPLE_SINT + 1;
    NONRETAIN_OUT.SIMPLE_STRING := ANY_TO_STRING(NONRETAIN_OUT.SIMPLE_DINT) + ' ' + ANY_TO_STRING(NONRETAIN_OUT.SIMPLE_TIME);
    NONRETAIN_OUT.SIMPLE_TIME := NONRETAIN_OUT.SIMPLE_TIME + PULSE_TIME;
    NONRETAIN_OUT.SIMPLE_UDINT := NONRETAIN_OUT.SIMPLE_UDINT + 1;
    NONRETAIN_OUT.SIMPLE_UINT := NONRETAIN_OUT.SIMPLE_UINT + 1;
    NONRETAIN_OUT.SIMPLE_ULINT := NONRETAIN_OUT.SIMPLE_ULINT + 1;
    NONRETAIN_OUT.SIMPLE_ULINT := NONRETAIN_OUT.SIMPLE_ULINT + 1;
    NONRETAIN_OUT.SIMPLE_WORD := NONRETAIN_OUT.SIMPLE_WORD + 1;

    AUTO1_OUT.SIMPLE_BOOL := NOT AUTO1_OUT.SIMPLE_BOOL;
    AUTO1_OUT.SIMPLE_BYTE := AUTO1_OUT.SIMPLE_BYTE + 1;
    AUTO1_OUT.SIMPLE_DATE := ANY_TO_DATE(1445385600 + AUTO1_OUT.SIMPLE_DINT * 86400);
    AUTO1_OUT.SIMPLE_DINT := AUTO1_OUT.SIMPLE_DINT + 1;
    AUTO1_OUT.SIMPLE_DWORD := AUTO1_OUT.SIMPLE_DWORD + 1;
    AUTO1_OUT.SIMPLE_INT := AUTO1_OUT.SIMPLE_INT + 1;
    AUTO1_OUT.SIMPLE_LINT := AUTO1_OUT.SIMPLE_LINT + 1;
    AUTO1_OUT.SIMPLE_LREAL := AUTO1_OUT.SIMPLE_LREAL + 1.1;
    AUTO1_OUT.SIMPLE_LWORD := AUTO1_OUT.SIMPLE_LWORD + 1;
    AUTO1_OUT.SIMPLE_REAL := AUTO1_OUT.SIMPLE_REAL + 1.1;
    AUTO1_OUT.SIMPLE_SINT := AUTO1_OUT.SIMPLE_SINT + 1;
    AUTO1_OUT.SIMPLE_STRING := ANY_TO_STRING(AUTO1_OUT.SIMPLE_DINT) + ' ' + ANY_TO_STRING(AUTO1_OUT.SIMPLE_TIME);
    AUTO1_OUT.SIMPLE_TIME := AUTO1_OUT.SIMPLE_TIME + PULSE_TIME;
    AUTO1_OUT.SIMPLE_UDINT := AUTO1_OUT.SIMPLE_UDINT + 1;
    AUTO1_OUT.SIMPLE_UINT := AUTO1_OUT.SIMPLE_UINT + 1;
    AUTO1_OUT.SIMPLE_ULINT := AUTO1_OUT.SIMPLE_ULINT + 1;
    AUTO1_OUT.SIMPLE_ULINT := AUTO1_OUT.SIMPLE_ULINT + 1;
    AUTO1_OUT.SIMPLE_WORD := AUTO1_OUT.SIMPLE_WORD + 1;

    AUTO2_OUT.SIMPLE_BOOL := AUTO1_OUT.SIMPLE_BOOL;
    AUTO2_OUT.SIMPLE_BYTE := AUTO1_OUT.SIMPLE_BYTE;
    AUTO2_OUT.SIMPLE_DATE := AUTO1_OUT.SIMPLE_DATE;
    AUTO2_OUT.SIMPLE_DINT := AUTO1_OUT.SIMPLE_DINT;
    AUTO2_OUT.SIMPLE_DWORD := AUTO1_OUT.SIMPLE_DWORD;
    AUTO2_OUT.SIMPLE_INT := AUTO1_OUT.SIMPLE_INT;
    AUTO2_OUT.SIMPLE_LINT := AUTO1_OUT.SIMPLE_LINT;
    AUTO2_OUT.SIMPLE_LREAL := AUTO1_OUT.SIMPLE_LREAL;
    AUTO2_OUT.SIMPLE_LWORD := AUTO1_OUT.SIMPLE_LWORD;
    AUTO2_OUT.SIMPLE_REAL := AUTO1_OUT.SIMPLE_REAL;
    AUTO2_OUT.SIMPLE_SINT := AUTO1_OUT.SIMPLE_SINT;
    AUTO2_OUT.SIMPLE_STRING := AUTO1_OUT.SIMPLE_STRING;
    AUTO2_OUT.SIMPLE_TIME := AUTO1_OUT.SIMPLE_TIME;
    AUTO2_OUT.SIMPLE_UDINT := AUTO1_OUT.SIMPLE_UDINT;
    AUTO2_OUT.SIMPLE_UINT := AUTO1_OUT.SIMPLE_UINT;
    AUTO2_OUT.SIMPLE_ULINT := AUTO1_OUT.SIMPLE_ULINT;
    AUTO2_OUT.SIMPLE_ULINT := AUTO1_OUT.SIMPLE_ULINT;
    AUTO2_OUT.SIMPLE_WORD := AUTO1_OUT.SIMPLE_WORD;
END_IF;

END_FUNCTION_BLOCK
